FUNCTION_BLOCK TestPID
VAR_INPUT
END_VAR
VAR_OUTPUT
END_VAR
VAR
	Ramp: Ramp;
	PidController: PidController;
	Target: lreal := 1;
END_VAR

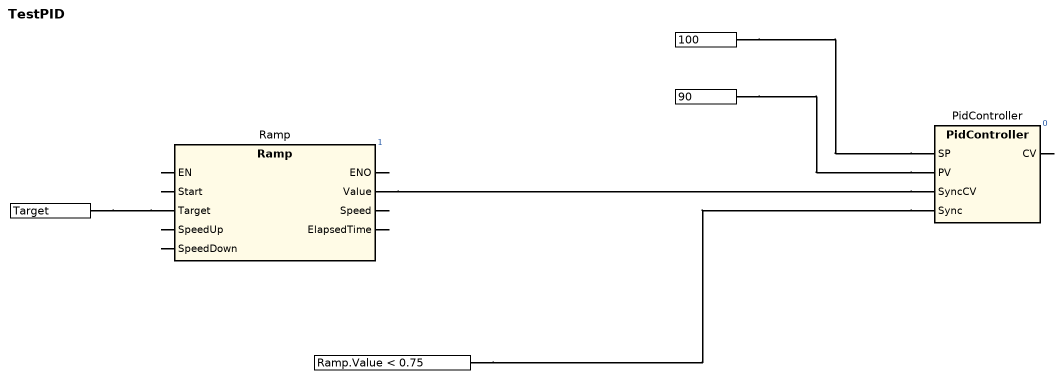
PidController(SP := 100, PV := 90, SyncCV := Ramp.Value, Sync := Ramp.Value < 0.75);
Ramp(Target := Target);

END_FUNCTION_BLOCK

(* stored: Version 1.1.0.1, ProductVersion 3.1.4024.6
   POU TestPID: Id {b7cad349-a42d-4524-bebf-01a02dbcf9d1}, SpecialFunc None *)
